FUNCTION_BLOCK DAerationLogic_HMI (* Service Interface Function Block Type *)
  (* Standard: 61499-2 *)
  (* Version 0.0, 10/24/2023, SESA685388, Schneider Electric, template *)
  PACKAGE SE.Nereda;
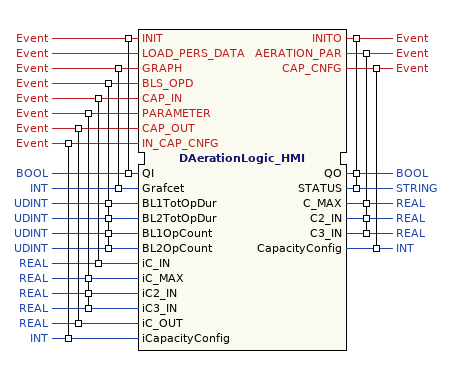
  EVENT_INPUT
    INIT WITH QI;
    LOAD_PERS_DATA;
    GRAPH WITH Grafcet;
    BLS_OPD WITH BL1TotOpDur, BL2TotOpDur, BL1OpCount, BL2OpCount;
    CAP_IN WITH iC_IN;
    PARAMETER WITH iC_MAX, iC2_IN, iC3_IN;
    CAP_OUT WITH iC_OUT;
    IN_CAP_CNFG WITH iCapacityConfig;
  END_EVENT
  EVENT_OUTPUT
    INITO WITH QO, STATUS;
    AERATION_PAR WITH C_MAX, C2_IN, C3_IN;
    CAP_CNFG WITH CapacityConfig;
  END_EVENT
  VAR_INPUT
    QI : BOOL;
    Grafcet : INT;
    BL1TotOpDur : UDINT;
    BL2TotOpDur : UDINT;
    BL1OpCount : UDINT;
    BL2OpCount : UDINT;
    iC_IN : REAL;
    iC_MAX : REAL;
    iC2_IN : REAL;
    iC3_IN : REAL;
    iC_OUT : REAL;
    iCapacityConfig : INT;
  END_VAR
  VAR_OUTPUT
    QO : BOOL; (* Event Output Qualifier *)
    STATUS : STRING; (* Service Status *)
    C_MAX : REAL;
    C2_IN : REAL;
    C3_IN : REAL;
    CapacityConfig : INT;
  END_VAR
  SERVICE /
    SEQUENCE 
    END_SEQUENCE
  END_SERVICE
END_FUNCTION_BLOCK
